{attribute addProperty BoxType "EK1122-0000-0018"}
{attribute addProperty Id "Beckhoff_EK13xxsub_EK1100EK1100_179A0949162A_0001_EK1300_0000_0017EK1300_D787878A486"}
{attribute addProperty CRC "728523881"}
{attribute addProperty SizeInBites "64"}
{attribute addProperty SizeInBytes "8"}
TYPE Beckhoff_EK13xxEK1122_2B6C6469 EXTENDS EK1122_179A0949 :
STRUCT
	{attribute addProperty Name "Beckhoff_EK13xxsub_EK1100"}
	Beckhoff_EK13xxsub_EK1100 : EK1100_179A0949;
	{attribute addProperty Name "A_0001_EK1300_0000_0017"}
	A_0001_EK1300_0000_0017 : EK1300_D787878A;
END_STRUCT
END_TYPE

(* stored: Version 1.2.0.0, ProductVersion 3.1.4024.9
   DUT Beckhoff_EK13xxEK1122_2B6C6469: Id {9ccf1774-4095-4917-b232-26612a71b065} *)
